(* CODESYS project SNDLTN_MQTT.library
   Title: SNDLTN_MQTT
   Author: S. Verbeek
   Version: 1.2.200929
   Company: Sandolution

Project tree, tasks and I/O mapping:
  libraries: CAA Net Base Services, * (CAA Technical Workgroup); Standard, * (System); CAA Memory, * (CAA Technical Workgroup); CAA Tick, 3.0.0.0 (3S - Smart Software Solutions GmbH); CAA TickUtil, 3.0.0.2 (CAA Technical Workgroup); CAA Types, 3.0.0.2 (3S - Smart Software Solutions GmbH)
  Constants/
    global variables MQTT_Properties
  Enums/
    data type MQTT_eState
    data type MQTT_eError
  Function Blocks/
    function block MQTT_Client [ST]: M_AppendOutputByte, M_AppendOutputString, M_AppendOutputLengthAndString, Main, M_AppendOutputWord
    function block MQTT_DecodeLength [ST]
    function block MQTT_EncodeLength [ST]
  Functions/
    function MQTT_RandomNumber [ST]
  Structs/
  Variables/
  program ChangeLog [ST]
*)

// Enums/MQTT_eState
{attribute 'qualified_only'}
TYPE MQTT_eState :
(
	Error := -1,
	Disabled := 0,					//Wait for enable
	                    		
	//TCP               		
	TCP_Connect := 1,				//Make TCP connection
	
	//Broker
	BrokerConnect := 5,				//Send connect to broker
	BrokerConnectAck := 6,			//Analyze connection acknowledgement 
	BrokerDisconnect := 8,			//Send disconnect to broker
	
	//Default
	Idle := 10,						//Wait for pub,sub or disconnect
	
	//Pub/Sub
	Subscribe := 20,				//Send subscribe message
	SubscribeAck := 21,				//Wait for acknowledgement from broker
	SubscribeReceive := 25,			//Incoming message
	Publish := 30					//Publish a message to topic

	

);
END_TYPE

// Enums/MQTT_eError
{attribute 'qualified_only'}
{attribute 'to_string'}
TYPE MQTT_eError :
(
	NoError 					:= 0,		//No Error
	
	//2000-2999 : MQTT ERRORS
	
	//Custom errors
	InvalidMQTT					:= 2000,	//Invalid MQTT response
	BufferOverflow				:= 2001,	//Overflow from method
	ConnectionLost				:= 2002,	//Connection with server lost
	TimeOut						:= 2003,	//Program time out, pub/sub no response
                            	
	//Broker responses      	
	RefusedProtocolVersion		:= 2010,	//Wrong protocol version
	RefusedIdentifier			:= 2011,	//Identifier rejected
	RefusedUserPass				:= 2012,	//Server unavailable
	RefusedAuthorization		:= 2013,	//Authorization failed
	ServerUnavailable			:= 2014,	//Server not available	
		
	//NBS errors (ported from 6001-6099)
	NBS_TimeOut 				:= 2100,	//Time limit exceeded
	NBS_InvalidAddress			:= 2101,	//Address invalid
	NBS_InvalidHandle			:= 2102,	//Handle invalid
	NBS_InvalidPointer			:= 2103,	//Data pointer invalid
	NBS_InvalidSize				:= 2104,	//Data size invalid
	NBS_ReceiveUDP				:= 2105,	//Error receiving data via UDP
	NBS_SendUDP					:= 2106,	//Error sending data via UDP
	NBS_SentIncompleteUDP		:= 2107,	//Not all data is sent.
	NBS_OpenUDP					:= 2108,	//Couldn't open UDP connection
	NBS_CloseUDP				:= 2109,	//Couldn't close UDP connection
	NBS_SendTCP					:= 2110,	//Error sending data via TCP
	NBS_ReceiveTCP				:= 2111,	//Error receiving data via TCP
	NBS_OpenTCP					:= 2112,	//Couldn't open TCP connection
	NBS_ConnectTCP				:= 2113,	//Couldn't connect TCP connection
	NBS_CloseTCP				:= 2114,	//Couldn't close TCP connection
	NBS_ServerTCP				:= 2115,	//Server error TCP
	NBS_WrongParameter			:= 2116,	//Wrong parameters entered
	NBS_Unknown					:= 2117		//Not specified
);
END_TYPE

// Constants/MQTT_Properties
{attribute 'qualified_only'}
VAR_GLOBAL CONSTANT
	uiMQTTMaxTopicSize			:UINT := 512;
	uiMQTTMaxMessageSize		:UINT := 4096;
	
	byMQTTProtocolLevel			:BYTE := 4;				//Version 3.1.1 - OASIS
END_VAR

// ChangeLog
PROGRAM ChangeLog
VAR
END_VAR

//Library for MQTT communication with other systems.

//V1.2.200929
//Compiler fixes for error C0327.
//Compatibility with x64 > use of __UXINT for szSize in MQTT_Client and for TICKS in MQTT_RandomNumber.
//Renamed sLastWillRetain to xLastWillRetain.

//V1.2.200714
//Fixed bug where xError wasn't reset to false when xConnect was made false (FB_TCPClient not deactivated).

//V1.2
//Update to compiler 3.5.14.40.
//Fixed bug for TCP errors which were in range 0-99 instead of 2200-2299.
//Updated state values.
//Added TCP_Client error handler.

//V1.1 - Feb 2019
//Changed constants into properties.
//Added conditionalshow attributes.

//V1.0 - Jan 2019:
//Integration of function blocks.

END_PROGRAM

// Function Blocks/MQTT_Client

{attribute 'conditionalshow_all_locals'}
FUNCTION_BLOCK MQTT_Client
VAR_INPUT
	//General
	xEnable							:BOOL;							//Enable FB
	xConnect						:BOOL;							//Start connection
	tTimeOut						:TIME := T#1S;					//Time out of functions and connections
	                            	                            	
	//Broker connection         	                            	
	sBrokerIP						:STRING(15) := '192.168.1.10';	//Address of broker
	uiBrokerPort					:UINT := 1883;					//Port of broker
	sBrokerUser						:STRING(64);					//Username to login on broker - optional
	sBrokerPass						:STRING(64);					//Password to login on broker - optional
	
	//Subscribe
	xSubscribe						:BOOL;							//Subscribe to topic
	sSubscribeTopic					:STRING(MQTT_Properties.uiMQTTMaxTopicSize) := 'in';		//Subscribe to topic
	                            	
	//Publish                   	
	xPublish						:BOOL;							//Publish message on topic
	sPublishTopic					:STRING(MQTT_Properties.uiMQTTMaxTopicSize) := 'out';	//Publish to topic
	sPublishMessage					:STRING(MQTT_Properties.uiMQTTMaxMessageSize) := 'HelloWorld';	//Message to publish
	xPublishRetain					:BOOL;							//Tell broker to retain message
	
	//Last Will and Testament
	sLastWillTopic					:STRING(MQTT_Properties.uiMQTTMaxTopicSize);		//Last will to broker		
	sLastWillMessage				:STRING(MQTT_Properties.uiMQTTMaxMessageSize);	//Last will message
 	xLastWillRetain					:BOOL;							//Tell broker to retain message
END_VAR                                                         	
VAR_OUTPUT                                                      	
	//General                                                   	
	eState							:MQTT_eState;					//Actual state
	                                                            	
	//Error                                                     	
	xError							:BOOL;							//Error occured
	eErrorID						:MQTT_eError;					//Error information
	                                                            	
	//Status                                                    	
	xConnected						:BOOL;							//Connection succesfull
	xSubscribed						:BOOL;							//Subscribed succesfully
	xPublished						:BOOL;							//Published succesfully
	
	//Subscribe
	xSubscriptionNewMessage			:BOOL;							//New message received
	sSubscriptionTopic				:STRING(MQTT_Properties.uiMQTTMaxTopicSize);		//Incoming subscription message - topic
	sSubscriptionMessage			:STRING(MQTT_Properties.uiMQTTMaxMessageSize);	//Incoming subscription message - message
END_VAR

VAR
	//General
	eStateRequested					:MQTT_eState;					//Next step in state machine
	eStateActive					:MQTT_eState;					//Active state
	
	//Error
	xError_int						:BOOL;							//Error occured
	eErrorID_int					:MQTT_eError;					//Error information
	
	//Input mems
	sBrokerIP_int					:STRING(15) := '192.168.1.10';	//Address of broker
	uiBrokerPort_int				:UINT := 1883;					//Port of broker
	xConnect_old					:BOOL;							//Store connect trigger
	xSubscribe_old					:BOOL;							//Store subscribe trigger
	xPublish_old					:BOOL;							//Store publish trigger
	                                
	//Outputs                        
	xConnected_int					:BOOL;							//Connection succesfull
	xSubscribed_int					:BOOL;							//Subscribed succesfully
	xPublished_int					:BOOL;							//Published succesfully

	//Incoming message
	xSubscriptionMessageAccepted	:BOOL;							//New message accepted
	xSubscriptionMessageRejected	:BOOL;							//New message rejected
	sSubscriptionTopic_int			:STRING(MQTT_Properties.uiMQTTMaxTopicSize);	//Incoming subscription message - topic
	sSubscriptionMessage_int		:STRING(MQTT_Properties.uiMQTTMaxMessageSize);	//Incoming subscription message - message
		
	//Function blocks
	//Data processing
	FB_DecodeLength					:MQTT_DecodeLength;				//Decode according to MQTT standards
	FB_EncodeLength					:MQTT_EncodeLength;				//Encode according to MQTT standards
	
	//TCP
	FB_TCPClient					:NBS.TCP_Client;				//TCP connection
	
	//Read data
	FB_TCPRead						:NBS.TCP_Read;					//Read TCP
	xTCPRead_Reset					:BOOL;							//Reset read FB
	uxiTCPRead_Size					:__UXINT;						//Store amount of bytes read
	abyTCPRead_Data_int				:ARRAY[0..MQTT_Properties.uiMQTTMaxMessageSize] OF BYTE;	//Read input buffer
	abyTCPRead_Data					:ARRAY[0..MQTT_Properties.uiMQTTMaxMessageSize] OF BYTE;	//Read input buffer > Stored 
	//Received subscribe message
	uiTPCRead_TopicStart			:UINT;							//Start of received subscribe topic
	uiTPCRead_TopicLength			:UINT;							//Length of received subscribe topic 
	uiTPCRead_MessageStart			:UINT;							//Start of received subscribe message
	uiTPCRead_MessageLength			:UINT;							//Length of received subscribe message

	//Write data
	FB_TCPWrite						:NBS.TCP_Write;					//Write TCP
	abyTCPWrite_Data				:ARRAY[0..MQTT_Properties.uiMQTTMaxMessageSize] OF BYTE;	//Write output buffer
	uiTCPWrite_Index				:UINT;							//Active position of write buffer

	wTCPWrite_Ident					:WORD;							// Message identifier according to MQTT standards

	//Timeout
	TON_TimeOut						:TON;							//Timer to guard active function
	
	//Internal	
	xMethodOverflow					:BOOL;							//Overflow occured while using method
	xMethodOverflow_mem				:BOOL;							//Mem overflow
	idx								:WORD;							//Loop variable (FOR)
	byx								:BYTE;							//Helper for payload
	
END_VAR

//Execute function block
IF xEnable THEN
	Main();
	
//Reset outputs
ELSE
	//General
	eState := MQTT_eState.Disabled;
	eStateRequested := MQTT_eState.Disabled;
	xError := FALSE;
	eErrorID := MQTT_eError.NoError;
	
	//Status
	xConnected := FALSE;
	xSubscribed := FALSE;
	xPublished := FALSE;
	
	//Subscribe
	xSubscriptionNewMessage := FALSE;
	sSubscriptionTopic := '';
	sSubscriptionMessage := '';
END_IF

{attribute 'conditionalshow'}
METHOD M_AppendOutputByte
VAR_INPUT
	byOutput:					BYTE;							(* Byte to insert *)
END_VAR

VAR_OUTPUT
	xOverflow:					BOOL;							(* Output buffer length exceeded *)
END_VAR
(* Append byte to output buffer, if possible *)

xOverflow := uiTCPWrite_Index >= SIZEOF(abyTCPWrite_Data);
IF NOT xOverflow THEN
	abyTCPWrite_Data[uiTCPWrite_Index] := byOutput;
	uiTCPWrite_Index := uiTCPWrite_Index + 1; 
END_IF;
END_METHOD

{attribute 'conditionalshow'}
METHOD M_AppendOutputString
VAR_INPUT
	sOutput					:STRING(MQTT_Properties.uiMQTTMaxMessageSize);							(* String to insert *)
END_VAR

VAR_OUTPUT
	xOverflow				:BOOL;							(* Output buffer length exceeded *)
END_VAR

VAR
	uiLength				:UINT;							(* Length of string to append *)
END_VAR
(* Append byte to output buffer, if possible *)

uiLength := INT_TO_UINT(LEN(sOutput));

xOverflow := uiTCPWrite_Index + uiLength >= SIZEOF(abyTCPWrite_Data);
IF NOT xOverflow THEN
	MEM.MemMove( 
		pSource:= ADR(sOutput), 
		pDestination:= ADR(abyTCPWrite_Data[uiTCPWrite_Index]), 
		uiNumberOfBytes:= uiLength
	);
	uiTCPWrite_Index := uiTCPWrite_Index + uiLength; 
END_IF;
END_METHOD

{attribute 'conditionalshow'}
METHOD M_AppendOutputLengthAndString
VAR_INPUT
	sOutput:					STRING;							(* Byte to insert *)
END_VAR

VAR_OUTPUT
	xOverflow:					BOOL;							(* Output buffer length exceeded *)
END_VAR

VAR
	uiLength:					UINT;							(* Length of string to append *)
END_VAR
(* Append string and length of string to output buffer, if possible *)

(* Length of string *)
uiLength := INT_TO_UINT(LEN(sOutput));

(* Test if possbile to append string and one word for length *)
xOverflow := uiTCPWrite_Index + uiLength + 2 >= SIZEOF(abyTCPWrite_Data);

(* Append data to output buffer *)
IF NOT xOverflow THEN
	(* Append length of string *)
	abyTCPWrite_Data[uiTCPWrite_Index] := MEM.HighByte(uiLength);
	uiTCPWrite_Index := uiTCPWrite_Index + 1; 
	abyTCPWrite_Data[uiTCPWrite_Index] := MEM.LowByte(uiLength);
	uiTCPWrite_Index := uiTCPWrite_Index + 1;
 
	(* Append contents of string *)
	MEM.MemMove( 
		pSource:= ADR(sOutput), 
		pDestination:= ADR(abyTCPWrite_Data[uiTCPWrite_Index]), 
		uiNumberOfBytes:= uiLength
	);
	uiTCPWrite_Index := uiTCPWrite_Index + uiLength; 
END_IF;
END_METHOD

ACTION Main:
{warning disable C0327}

//Change actual state (cycle sensitive)
IF eStateRequested <> eStateActive THEN
	eStateActive := eStateRequested;
END_IF
 

//State machine
CASE eStateActive OF

	//************************************************************************************************************************************************ERROR
	MQTT_eState.Error:	
	
		//Wait for reset condition
		IF NOT xConnect THEN
			xError_int := FALSE;
			eErrorID_int := MQTT_eError.NoError;
			xConnect_old := FALSE; //Restart connection
			eStateRequested := MQTT_eState.Disabled;
		END_IF
	
	//************************************************************************************************************************************************DISABLED
	MQTT_eState.Disabled: 	
		
		//Disable timeout
		TON_TimeOut.PT := T#0MS;
		
		//(re)start connection
		IF xConnect AND NOT xConnect_old THEN	//Flank
			xConnect_old := TRUE;
			sBrokerIP_int := sBrokerIP;
			uiBrokerPort_int := uiBrokerPort;
			eStateRequested := MQTT_eState.TCP_Connect;
		END_IF
		
		//Remove all status
		xConnected_int := FALSE;
		xSubscribed_int := FALSE;
		xPublished_int := FALSE;
		
		//Remove any subscribed messages
		xSubscriptionMessageAccepted := FALSE;
		xSubscriptionMessageRejected := FALSE;
		sSubscriptionTopic_int := '';
		sSubscriptionMessage_int := '';

	//************************************************************************************************************************************************TCP CONNECT
	MQTT_eState.TCP_Connect:		
		
		//Set TB timeout
		TON_TimeOut.PT := tTimeOut;
		
		//TCP Client is automatically started via state machine input on execute
		
		//Check for existing connection
		IF FB_TCPClient.hConnection <> 0 AND xConnected_int THEN
			eStateRequested := MQTT_eState.BrokerConnect;
			
		//Check for error
		ELSIF TON_TimeOut.Q OR FB_TCPClient.xError THEN
			xError_int := TRUE;
			IF FB_TCPClient.xError THEN
				eErrorID_int := FB_TCPClient.eError;
			ELSE
				eErrorID_int := MQTT_eError.TimeOut;
			END_IF
			//State
			eStateRequested := MQTT_eState.Error;	
		END_IF
		
	//************************************************************************************************************************************************BROKER CONNECT
	MQTT_eState.BrokerConnect: 

		//Empty total buffer
		uiTCPWrite_Index := 0;
		MEM.MemFill(ADR(abyTCPWrite_Data), SIZEOF(abyTCPWrite_Data), 0);
		
		//Add byte
		M_AppendOutputByte(byOutput := 16);
		
		//Calculate the length: Length must be 10 (for variable header) + Payload (We use 10 bytes client ID) *)
		//20: 10byte variable header and 10byte client Id *)
		// "2+..." because legth of that string has to be added if string is used *)
		FB_EncodeLength(
			udiLengthRemaining:= TO_UINT(20 + (2+LEN(sBrokerUser)) * TO_INT(sBrokerUser <> '') + (2+LEN(sBrokerPass)) * TO_INT(sBrokerPass <> '') 
								+ (2+LEN(sLastWillTopic)) * TO_INT(sLastWillTopic <> '') + (2+LEN(sLastWillMessage)) * TO_INT(sLastWillMessage <> ''))
		);
			
		//Load remaining length info
		FOR idx := 0 TO FB_EncodeLength.uiLengthBytesCount - 1 DO
			M_AppendOutputByte(byOutput:= FB_EncodeLength.abyLengthBytes[idx]);
		END_FOR;

		//Protocol header
		M_AppendOutputLengthAndString(sOutput := 'MQTT');
		
		//Protocol level
		M_AppendOutputByte(byOutput:= MQTT_Properties.byMQTTProtocolLevel);
	
		//Connect flags 0: Reserved; 1: Clean Session, 2: Will Flag, 3+4: Will QoS, 5: Will Retain, 6: Password Flag, 7: Username Flag
		byx := SHL(TO_BYTE(sLastWillTopic <> ''), 2)
						OR SHL(TO_BYTE(xLastWillRetain), 5)
						OR SHL(TO_BYTE(sBrokerPass <> ''), 6)
						OR SHL(TO_BYTE(sBrokerUser <> ''), 7);
		M_AppendOutputByte(byOutput := byx);

		//Keep alive (not implemented yet)
		M_AppendOutputWord(wOutput := 0);

		//Generate client ID
		M_AppendOutputWord(wOutput := 8);	
		FOR idx := 2 TO 9 DO
			M_AppendOutputByte(byOutput := TO_BYTE(MQTT_RandomNumber(65,90)));		//Client name (ASCII 65-90) according to MQTT specs
		END_FOR;
		
		//Reset mem
		xMethodOverflow_mem := FALSE;
		
		//Add last will topic
		IF sLastWillTopic <> '' THEN
			M_AppendOutputLengthAndString(sOutput := sLastWillTopic, xOverflow => xMethodOverflow);
		END_IF
		IF xMethodOverflow THEN xMethodOverflow_mem := TRUE; END_IF
		
		//Add last will message
		IF sLastWillMessage <> '' THEN
			M_AppendOutputLengthAndString(sOutput := sLastWillMessage, xOverflow => xMethodOverflow);
		END_IF
		IF xMethodOverflow THEN xMethodOverflow_mem := TRUE; END_IF
		
		//Add username
		IF sBrokerUser <> '' THEN
			M_AppendOutputLengthAndString(sOutput := sBrokerUser, xOverflow => xMethodOverflow);
		END_IF
		IF xMethodOverflow THEN xMethodOverflow_mem := TRUE; END_IF
		
		//Add password
		IF sBrokerPass <> '' THEN
			M_AppendOutputLengthAndString(sOutput := sBrokerPass, xOverflow=> xMethodOverflow);
		END_IF
		IF xMethodOverflow THEN xMethodOverflow_mem := TRUE; END_IF
		
		//Check for overflow
		IF xMethodOverflow_mem THEN
			xError_int := TRUE;
			eErrorID_int := MQTT_eError.BufferOverflow;
			//State
			eStateRequested := MQTT_eState.Error;	
		ELSE
			//Transfer data to FB
			FB_TCPWrite.szSize := LIMIT(0,uiTCPWrite_Index,SIZEOF(abyTCPWrite_Data));
			FB_TCPWrite.pData := ADR(abyTCPWrite_Data);
			
			//Start writing
			TON_TimeOut.PT := tTimeOut;
			FB_TCPWrite.xExecute := TRUE;
		END_IF
		
		//Wait for done / error
		IF FB_TCPWrite.xDone AND NOT FB_TCPWrite.xError THEN
			FB_TCPWrite.xExecute := FALSE;
			uxiTCPRead_Size := 0;
			eStateRequested := MQTT_eState.BrokerConnectAck;
		ELSIF FB_TCPWrite.xError OR TON_TimeOut.Q THEN
			xError_int := TRUE;
			IF FB_TCPWrite.xError THEN
				eErrorID_int := FB_TCPWrite.eError;
			ELSE
				eErrorID_int := MQTT_eError.TimeOut;
			END_IF
			//State
			FB_TCPWrite.xExecute := FALSE;	
			eStateRequested := MQTT_eState.Error;	
		END_IF

	//************************************************************************************************************************************************BROKER ACK
	MQTT_eState.BrokerConnectAck: 
		
		//Set TB timeout
		TON_TimeOut.PT := T#1S;
		
		//Incoming message
		IF FB_TCPRead.xReady AND NOT FB_TCPRead.xError THEN
			
			//Reset read FB
			xTCPRead_Reset := TRUE;
			
			//Disable timeout
			TON_TimeOut.PT := T#0MS;
			
			//Check response from broker
			CASE abyTCPRead_Data[3] OF
				0: // Accepted
					IF abyTCPRead_Data[0] = 32 THEN
						eStateRequested := MQTT_eState.Idle;
					ELSE
						xError_int := TRUE;
						eErrorID_int := MQTT_eError.InvalidMQTT;
					END_IF
					
				1:	//Protocol version
					xError_int := TRUE;
					eErrorID_int := MQTT_eError.RefusedProtocolVersion;
					
				2:	//Identifier
					xError_int := TRUE;
					eErrorID_int := MQTT_eError.RefusedIdentifier;

				3:	//Server unavailable
					xError_int := TRUE;
					eErrorID_int := MQTT_eError.ServerUnavailable;

				4:	//Username / password
					xError_int := TRUE;
					eErrorID_int := MQTT_eError.RefusedUserPass;

				5:	//Not authorized
					xError_int := TRUE;
					eErrorID_int := MQTT_eError.RefusedAuthorization;

			END_CASE
		
		//Error occured
		ELSIF FB_TCPRead.xError OR (FB_TCPRead.xDone AND uxiTCPRead_Size=0) OR TON_TimeOut.Q THEN
			//Reset read FB
			xTCPRead_Reset := TRUE;
			
			xError_int := TRUE;
			IF FB_TCPRead.xError THEN
				eErrorID_int := FB_TCPRead.eError;
			ELSE
				eErrorID_int := MQTT_eError.TimeOut;
			END_IF
			//State
			eStateRequested := MQTT_eState.Error;	
		END_IF		
		
	
	//************************************************************************************************************************************************BROKER DISCONNECT
	MQTT_eState.BrokerDisconnect: 
		
		//Set TB timeout
		TON_TimeOut.PT := tTimeOut;
		
		//Empty total buffer
		uiTCPWrite_Index := 0;
		MEM.MemFill(ADR(abyTCPWrite_Data), SIZEOF(abyTCPWrite_Data), 0);
		
		//Prepare data
		abyTCPWrite_Data[0] := 16#E0;		//MQTT Control Packet Type - disconnect
		FB_TCPWrite.pData := ADR(abyTCPWrite_Data);
		FB_TCPWrite.szSize := 2;
		
		//Start
		FB_TCPWrite.xExecute := TRUE;
		
		//Wait for done > reconnect
		IF FB_TCPWrite.xDone AND NOT FB_TCPWrite.xError THEN
			xSubscribed_int := FALSE;	//Remove previous subscription
			xConnect_old := FALSE;		//Retrigger in disabled state
			FB_TCPWrite.xExecute := FALSE;
			eStateRequested := MQTT_eState.Disabled;
		//Error occured
		ELSIF FB_TCPWrite.xError OR TON_TimeOut.Q THEN
			//Write error
			xError_int := TRUE;
			IF FB_TCPWrite.xError THEN
				eErrorID_int := FB_TCPWrite.eError;
			ELSE
				eErrorID_int := MQTT_eError.TimeOut;
			END_IF
			//State
			FB_TCPWrite.xExecute := FALSE;	
			eStateRequested := MQTT_eState.Error;	
		END_IF
		
	//************************************************************************************************************************************************IDLE 
	//Wait for incoming message or subscribe / publish command
	MQTT_eState.Idle:	
	
		//Disable timeout
		TON_TimeOut.PT := T#0MS;
		
		//Remove old output
		xSubscriptionMessageAccepted:= FALSE;
		xSubscriptionMessageRejected := FALSE;

		//Check if data is received
		IF FB_TCPRead.xReady AND NOT FB_TCPRead.xError AND uxiTCPRead_Size > 0 THEN	
			//Reset read FB
			xTCPRead_Reset := TRUE;
			
			//New message received	
			eStateRequested := MQTT_eState.SubscribeReceive;	
		ELSIF FB_TCPRead.xError THEN
			//Reset read FB
			xTCPRead_Reset := TRUE;
			
			xError_int := TRUE;
			eErrorID_int := FB_TCPRead.eError;
			//State
			eStateRequested := MQTT_eState.Error;	
		END_IF			
        
		//Subscribe command
		IF xSubscribe AND NOT xSubscribe_old AND xConnected_int THEN
			xSubscribe_old := TRUE;
			eStateRequested := MQTT_eState.Subscribe;	
		//Break connection to remove subscribtion
		ELSIF NOT xSubscribe AND xSubscribed AND xConnected_int THEN
			eStateRequested := MQTT_eState.BrokerDisconnect;	
		END_IF
		
		//Publish command
		IF xPublish AND NOT xPublish_old AND xConnected_int THEN
			xPublish_old := TRUE;
			eStateRequested := MQTT_eState.Publish;	
		END_IF
				
		//Disconnect from broker
		IF NOT xConnect AND xConnected_int THEN
			eStateRequested := MQTT_eState.BrokerDisconnect;	
		END_IF
		
		//Communication lost
		IF NOT xConnected_int THEN
			xError_int := TRUE;
			eErrorID_int := MQTT_eError.ConnectionLost;
			eStateRequested := MQTT_eState.Error;
		END_IF

	//************************************************************************************************************************************************SUBSCRIBE
	MQTT_eState.Subscribe: 
	
		//Empty total buffer
		uiTCPWrite_Index := 0;
		MEM.MemFill(ADR(abyTCPWrite_Data), SIZEOF(abyTCPWrite_Data), 0);
		
		//Add control packet type
		M_AppendOutputByte(byOutput:= 16#80 OR 16#2);	//Packet type + reserved
		
		//Set length (Identifier + length + topic + qos)
		FB_EncodeLength(udiLengthRemaining:= TO_WORD(LEN(sSubscribeTopic)) + 5);
			
		//Set remaining length
		FOR idx := 0 TO FB_EncodeLength.uiLengthBytesCount - 1 DO
			M_AppendOutputByte(byOutput:= FB_EncodeLength.abyLengthBytes[idx]);
		END_FOR;

		//Message identifier
		wTCPWrite_Ident := wTCPWrite_Ident + 1;	//Increase one
		IF wTCPWrite_Ident = 0 THEN //Guard overflow / zero since this is invalid
			wTCPWrite_Ident := 1;
		END_IF
		M_AppendOutputWord(wOutput:= wTCPWrite_Ident);//Add to message
		
		//Reset mem
		xMethodOverflow_mem := FALSE;
		
		//Add topic name
		IF TO_UINT(LEN(sSubscribeTopic)) > 0 THEN
			M_AppendOutputLengthAndString(sOutput := sSubscribeTopic, xOverFlow => xMethodOverflow);
		END_IF
		IF xMethodOverflow THEN xMethodOverflow_mem := TRUE; END_IF
		
		IF xMethodOverflow_mem THEN
			xError_int := TRUE;
			eErrorID_int := MQTT_eError.BufferOverflow;
		ELSE
			//Add QoS > Always zero
			M_AppendOutputByte(byOutput := 0);	
			
			//Set data for writing
			FB_TCPWrite.pData := ADR(abyTCPWrite_Data);
			FB_TCPWrite.szSize := uiTCPWrite_Index;
			
			//Write data
			TON_TimeOut.PT := tTimeOut;	
			FB_TCPWrite.xExecute := TRUE;
		END_IF
		
		//Wait for done
		IF FB_TCPWrite.xDone AND NOT FB_TCPWrite.xError THEN
			FB_TCPWrite.xExecute := FALSE;
			eStateRequested := MQTT_eState.SubscribeAck;
		ELSIF FB_TCPWrite.xError OR TON_TimeOut.Q THEN
			xError_int := TRUE;
			IF FB_TCPWrite.xError THEN
				eErrorID_int := FB_TCPWrite.eError;
			ELSE
				eErrorID_int := MQTT_eError.TimeOut;
			END_IF
			//State
			FB_TCPWrite.xExecute := FALSE;	
			eStateRequested := MQTT_eState.Error;			
		END_IF
		
			
	//************************************************************************************************************************************************SUBSCRIBE ACK	
	MQTT_eState.SubscribeAck: 

		//Set FB timeout
		TON_TimeOut.PT := tTimeOut;
		
		//Wait until ack received
		IF FB_TCPRead.xReady AND NOT FB_TCPRead.xError THEN		
			//Reset read FB
			xTCPRead_Reset := TRUE;
			
			//Disable timeout
			TON_TimeOut.PT := T#0MS;
			
			//Check response
			IF abyTCPRead_Data[uxiTCPRead_Size-1] < 16#80 THEN
				eStateRequested := MQTT_eState.Idle;
				xSubscribed_int := TRUE;
				uxiTCPRead_Size:=0;
			ELSE	
				xError_int := TRUE;
				eErrorID_int := MQTT_eError.InvalidMQTT;
			END_IF

		//Error occured
		ELSIF FB_TCPRead.xError OR (FB_TCPRead.xDone AND uxiTCPRead_Size=0) OR TON_TimeOut.Q THEN
			//Reset read FB
			xTCPRead_Reset := TRUE;
			
			xError_int := TRUE;
			IF FB_TCPRead.xError THEN
				eErrorID_int := FB_TCPRead.eError;
			ELSE
				eErrorID_int := MQTT_eError.TimeOut;
			END_IF
			//State
			eStateRequested := MQTT_eState.Error;	
		END_IF

	//************************************************************************************************************************************************SUBSCRIBED INCOMING
	MQTT_eState.SubscribeReceive: 
	
		//Disable timeout
		TON_TimeOut.PT := T#0MS;
		
		//Check remaining lenght
		FOR idx := 0 TO 3 DO
			FB_DecodeLength.abyLengthBytes[idx] := abyTCPRead_Data[idx+1];
		END_FOR
		FB_DecodeLength();

		//Get incoming topic name
		uiTPCRead_TopicStart := 1 + FB_DecodeLength.uiLengthBytesCount;	//Fixed header + remaining length
		uiTPCRead_TopicLength := MEM.PackBytesToWord(byHighByte:=abyTCPRead_Data[1+FB_DecodeLength.uiLengthBytesCount], byLowByte:=abyTCPRead_Data[2+FB_DecodeLength.uiLengthBytesCount]);
		
		//Get incoming message
		uiTPCRead_MessageStart := uiTPCRead_TopicStart + 2 + uiTPCRead_TopicLength;	//Fixed header + remaining length > + identifier + topic lenght
		uiTPCRead_MessageLength := TO_UINT(uxiTCPRead_Size) - uiTPCRead_MessageStart;	//Payload is last item in buffer
		
		//Check if topic and message are valid and fit strings, if not > reject message
		IF uiTPCRead_TopicLength <= MQTT_Properties.uiMQTTMaxTopicSize 
		AND uiTPCRead_MessageLength <= MQTT_Properties.uiMQTTMaxMessageSize THEN
			//Load buffer to output
			MEM.MemFill(ADR(sSubscriptionTopic_int), SIZEOF(sSubscriptionTopic_int), 0);	//Reset
			MEM.MemMove(ADR(abyTCPRead_Data[uiTPCRead_TopicStart+2]), ADR(sSubscriptionTopic_int), uiTPCRead_TopicLength);
	
			//Load buffer to output
			MEM.MemFill(ADR(sSubscriptionMessage_int), SIZEOF(sSubscriptionMessage_int), 0);
			MEM.MemMove(ADR(abyTCPRead_Data[uiTPCRead_MessageStart]), ADR(sSubscriptionMessage_int), uiTPCRead_MessageLength);
			
			//Done
			uxiTCPRead_Size := 0;
			
			//Received message (out)
			xSubscriptionMessageAccepted:= TRUE;
			
		//Reject message without notification
		ELSE
			//Done
			uxiTCPRead_Size := 0;
			
			//Reject message (out)
			xSubscriptionMessageRejected := TRUE;
		END_IF
				
		//State
		eStateRequested := MQTT_eState.Idle;	
			
	//************************************************************************************************************************************************PUBLISH
	MQTT_eState.Publish: 
		//Empty total buffer
		uiTCPWrite_Index := 0;
		MEM.MemFill(ADR(abyTCPWrite_Data), SIZEOF(abyTCPWrite_Data), 0);
		
		//Add 
		M_AppendOutputByte(byoutput:= 16#30 OR TO_BYTE(xPublishRetain));	//Publish MQTT Packet type
	
		//Calculate length > Length of header + Length of message + offset
		FB_EncodeLength(udiLengthRemaining:= TO_UDINT(LEN(sPublishTopic) + LEN(sPublishMessage)) + 2);
			
		//Remaining length
		FOR idx := 0 TO FB_EncodeLength.uiLengthBytesCount - 1 DO
			M_AppendOutputByte(byOutput:= FB_EncodeLength.abyLengthBytes[idx]);
		END_FOR
		
		//Reset mem
		xMethodOverflow_mem := FALSE;

		//Add topic to publish
		IF TO_UINT(LEN(sPublishTopic)) > 0 THEN
			M_AppendOutputLengthAndString(sPublishTopic, xOverflow=> xMethodOverflow);
		END_IF
		IF xMethodOverflow THEN xMethodOverflow_mem := TRUE; END_IF

		//Add message to publish
		IF TO_UINT(LEN(sPublishMessage)) > 0 THEN
			M_AppendOutputString(sPublishMessage, xOverflow=> xMethodOverflow);
		END_IF
		IF xMethodOverflow THEN xMethodOverflow_mem := TRUE; END_IF
		
		//Detect overflow of buffer
		IF xMethodOverflow_mem THEN
			xError_int := TRUE;
			eErrorID_int := MQTT_eError.BufferOverflow;
		ELSE
			//Prepare data
			FB_TCPWrite.pData := ADR(abyTCPWrite_Data);
			FB_TCPWrite.szSize := LIMIT(0, uiTCPWrite_Index, SIZEOF(abyTCPWrite_Data));
	
			//Write data			
			TON_TimeOut.PT := tTimeOut;
			FB_TCPWrite.xExecute := TRUE;
		END_IF
		
		//Wait for done or error
		IF FB_TCPWrite.xDone AND NOT FB_TCPWrite.xError THEN
			FB_TCPWrite.xExecute := FALSE;
			xPublished_int := TRUE;
			eStateRequested := MQTT_eState.Idle;
		ELSIF FB_TCPWrite.xError OR TON_TimeOut.Q THEN		
			xError_int := TRUE;
			IF FB_TCPWrite.xError THEN
				eErrorID_int := FB_TCPWrite.eError;
			ELSE
				eErrorID_int := MQTT_eError.TimeOut;
			END_IF
			//State
			FB_TCPWrite.xExecute := FALSE;	
			eStateRequested := MQTT_eState.Error;	
		END_IF
		
END_CASE

//Last: check TCP client itself outside program
IF NOT xError_int AND FB_TCPClient.xError THEN
	xError_int := TRUE;
	eErrorID_int := FB_TCPClient.eError;
END_IF

//Jump to error state if not catched in state machine
IF xError_int AND eStateRequested <> MQTT_eState.Error THEN
	eStateRequested := MQTT_eState.Error;
END_IF


//**************************************************************************
//Set IP address inside struct
FB_TCPClient.ipAddr.sAddr := sBrokerIP_int;

//Connect to server via TCP
FB_TCPClient(
	xEnable:= eStateActive > MQTT_eState.Disabled,
	xDone=> , 
	xBusy=> , 
	xError=> , 
	ipAddr:= , 
	uiPort:= uiBrokerPort_int, 
	eError=> , 
	xActive=> xConnected_int, 
	hConnection=> 
);
	
//Sent data to TCP
FB_TCPWrite(
	xExecute:= , 
	udiTimeOut:= TIME_TO_UDINT(tTimeOut), 
	xDone=> , 
	xBusy=> , 
	xError=> , 
	hConnection:= FB_TCPClient.hConnection, 
	szSize:= , 
	pData:= , 
	eError=>
);	

//Read data from TCP
FB_TCPRead(
	xEnable:= FB_TCPClient.xActive AND NOT xTCPRead_Reset,	//Reset if incoming message is processed 
	xDone=> , 
	xBusy=> , 
	xError=> , 
	hConnection:= FB_TCPClient.hConnection, 
	szSize:= SIZEOF(abyTCPRead_Data_int), 
	pData:= ADR(abyTCPRead_Data_int), 
	eError=> , 
	xReady=> , 
	szCount=>
);

//Reset TCP reset bit
IF xTCPRead_Reset THEN xTCPRead_Reset := FALSE; END_IF
	
//Store any message for processing
IF FB_TCPRead.xReady THEN
	FOR idx := 0 TO TO_UINT(FB_TCPRead.szCount) - 1 DO
		abyTCPRead_Data[idx] := abyTCPRead_Data_int[idx];
		uxiTCPRead_Size := TO_UDINT(FB_TCPRead.szCount);
	END_FOR
END_IF

//Guard timeout if activated
TON_TimeOut(IN:= TON_TimeOut.PT > T#0MS, PT:= );

//**************************************************************************
//Remove triggers
IF NOT xConnect AND xConnect_old THEN
	xConnect_old := FALSE;
END_IF

IF NOT xSubscribe AND xSubscribe_old THEN
	xSubscribe_old := FALSE;
	xSubscribed := FALSE;
END_IF

IF NOT xPublish AND xPublish_old THEN
	xPublish_old := FALSE;
	xPublished_int := FALSE;
END_IF

//**************************************************************************
//Transfer outputs from internal states
eState					:= eStateActive;
xError 					:= xError_int;
IF eErrorID_int < 6000 THEN
	eErrorID 			:= eErrorID_int;
ELSE
	eErrorID 			:= eErrorID_int - 3900; //NBS starts at 6000 > SNDLTN_MQTT at 2000 > -4000
END_IF
xConnected 				:= xConnected_int;
xSubscribed 			:= xSubscribed_int;
xPublished 				:= xPublished_int;
xSubscriptionNewMessage	:= xSubscriptionMessageAccepted;
sSubscriptionTopic		:= sSubscriptionTopic_int;
sSubscriptionMessage	:= sSubscriptionMessage_int;

{warning restore C0327}
END_ACTION

{attribute 'conditionalshow'}
METHOD M_AppendOutputWord
VAR_INPUT
	wOutput:					WORD;							(* Word to insert *)
END_VAR

VAR_OUTPUT
	xOverflow:					BOOL;							(* Output buffer length exceeded *)
END_VAR
(* Append word to output buffer, if possible. Highbyte first (MQTT standards) *)

xOverflow := uiTCPWrite_Index >= SIZEOF(abyTCPWrite_Data) - 1;
IF NOT xOverflow THEN
	abyTCPWrite_Data[uiTCPWrite_Index] := MEM.HighByte(wOutput);
	uiTCPWrite_Index := uiTCPWrite_Index + 1; 
	abyTCPWrite_Data[uiTCPWrite_Index] := MEM.LowByte(wOutput);
	uiTCPWrite_Index := uiTCPWrite_Index + 1; 
END_IF;
END_METHOD

END_FUNCTION_BLOCK

// Function Blocks/MQTT_DecodeLength
{attribute 'conditionalshow'}
FUNCTION_BLOCK MQTT_DecodeLength
VAR_INPUT
	abyLengthBytes				:ARRAY [0..3] OF BYTE;			//Length specification according to OASIS
END_VAR

VAR_OUTPUT
	udiLengthRemaining			:UDINT;							//Remaining length
	uiLengthBytesCount			:UINT;							//Amount of bytes in the length specification
END_VAR

//Check remaining length bytes
IF (abyLengthBytes[2] AND 16#80) <> 0 THEN
	udiLengthRemaining := udiLengthRemaining OR SHL(BYTE_TO_UDINT(abyLengthBytes[3] AND 16#7F), 21);
	uiLengthBytesCount := 4;
ELSIF (abyLengthBytes[1] AND 16#80) <> 0 THEN
	udiLengthRemaining := udiLengthRemaining OR SHL(BYTE_TO_UDINT(abyLengthBytes[2] AND 16#7F), 14);
	uiLengthBytesCount := 3;
ELSIF (abyLengthBytes[0] AND 16#80) <> 0 THEN
	udiLengthRemaining := udiLengthRemaining OR SHL(BYTE_TO_UDINT(abyLengthBytes[1] AND 16#7F), 7);
	uiLengthBytesCount := 2;
ELSE
	udiLengthRemaining := BYTE_TO_UDINT(abyLengthBytes[0] AND 16#7F);
	uiLengthBytesCount := 1;
END_IF;

END_FUNCTION_BLOCK

// Function Blocks/MQTT_EncodeLength
{attribute 'conditionalshow'}
FUNCTION_BLOCK MQTT_EncodeLength
VAR_INPUT
	udiLengthRemaining			:UDINT;							//Remaining length
END_VAR

VAR_OUTPUT
	abyLengthBytes				:ARRAY [0..3] OF BYTE;			//Length specification according to OASIS
	uiLengthBytesCount			:UINT;							//Amount of bytes in the length specification
END_VAR

VAR
	byEncoded					:BYTE;							//Encoded byte
	udiX						:UDINT;							//Temp variable
END_VAR

//Set all to zero before executing
uiLengthBytesCount := 0;
udiX := udiLengthRemaining;

//Check total length and split into array
REPEAT
	byEncoded := UDINT_TO_BYTE(udiX AND 16#7F);
	udiX := SHR(udiX, 7);
	IF udiX <> 0 THEN
		byEncoded := byEncoded OR 16#80;
	END_IF;
	abyLengthBytes[uiLengthBytesCount] := byEncoded;
	uiLengthBytesCount := uiLengthBytesCount + 1;
UNTIL 
	udiX = 0 
	AND uiLengthBytesCount < 4
END_REPEAT;

END_FUNCTION_BLOCK

// Functions/MQTT_RandomNumber
{attribute 'conditionalshow_all_locals'}
FUNCTION MQTT_RandomNumber : UDINT
VAR_INPUT
	udiLowLimit			:UDINT;		//Min number
	udiHighLimit		:UDINT;		//Max number
END_VAR
VAR
	uxiTick				:__UXINT;
	uxiShiftL			:__UXINT;
	uxiShiftR			:__UXINT;
	uxiTickShiftL		:__UXINT;
	uxiTickShiftR		:__UXINT;
	uxiTickModulo		:__UXINT;
END_VAR

uxiTick := TICKS.GetTick(0);  
uxiShiftL := (uxiTick MOD 17) + 1;	//prime number > avoid 0
uxiShiftR := (uxiTick MOD 7) + 1;	//prime number > avoid 0
uxiTickShiftL 	:= SHL(uxiTick, uxiShiftL);
uxiTickShiftR 	:= SHR(uxiTick, uxiShiftR);
uxiTickModulo	:= uxiTickShiftR MOD (udiHighLimit-udiLowLimit+1);
MQTT_RandomNumber := TO_UDINT(uxiTickModulo) + udiLowLimit;

END_FUNCTION
